(* CoDeSys 2.3 export: ERR_BLOCK.EXP *)

(* POU Alarm/ERR_BLOCK, ST *)
FUNCTION ERR_BLOCK : BOOL
VAR_INPUT
END_VAR
VAR
	i: INT := 1;
END_VAR
	ERR_BLOCK := FALSE;

	FOR i := 1 TO _ERR_Nums DO
		IF (glbErrors[i].LatchState OR glbErrors[i].State) AND glbErrors[i].Lock THEN
			ERR_BLOCK := TRUE;
		END_IF;
	END_FOR;
END_FUNCTION
